TYPE ST_AdjustmentProcessConfig :
STRUCT
    
    fAdjustTolerance : LREAL;// 同轴度调整阶段停止继续修正的容差。

    
    fQualifiedTolerance : LREAL;// 最终检测判定合格的容差。

    //==========================================================
    // Adjustment XY自动视觉闭环最大允许累计修正范围
    //
    // 单位：mm
    //
    // 基准位置：
    // GVL_PositionConfig.stAdjustment.stWork.X/Y
    //
    // 实际允许区域：
    // WorkX ± fMaxCorrectionX
    // WorkY ± fMaxCorrectionY
    //==========================================================
    fMaxCorrectionX : LREAL;
    fMaxCorrectionY : LREAL;

    
    nMaxAdjustCount : UINT;// 单轮最大视觉修正次数。

    // 每个逻辑Coax检测点首次失败后的额外检测次数和等待时间。
    nCoaxMaxRetryCount : UINT;
    tCoaxRetryDelay : TIME;

    
    nMaxReworkCount : UINT;// 最终检测失败后的最大返调次数。
END_STRUCT
END_TYPE

(* stored: Version 1.1.0.1, ProductVersion 3.1.4026.20
   DUT ST_AdjustmentProcessConfig: Id {03500fbb-864c-49b5-9597-9684309f44f6} *)
